KUKA KRL program: PutTmpFileHere.src

&ACCESS RVO1
&COMMENT
DEF PutTmpFileHere ( )

END
